{attribute 'qualified_only'}
VAR_GLOBAL
    {attribute 'TcLinkTo' := 'TIID^Device 1 (EtherCAT)^B940_009_R19_DRL_02_E0_EK1200^R19_DRL_02_E4_EK1122^Term 35 (EK1100)^B950-100H1-R02-PNL-01_E2^Channel 1^Input'}
    {attribute 'pytmc' := '
        pv: "DREAM:SL:STATUS",
        field: "DREAM Safety Loop Status",
        field: "ZNAM OPEN",
        field: "ONAM CLOSED"
    '}
    bSafetyLoopStatus AT %I* : BOOL;

        {attribute 'TcLinkTo' := 'TIID^Device 1 (EtherCAT)^B940_009_R19_DRL_02_E0_EK1200^R19_DRL_02_E4_EK1122^Term 35 (EK1100)^B950-100H1-R02-PNL-01_E1^Channel 1^Output'}
    {attribute 'pytmc' := '
        pv: "DREAM:SL:ENABLE",
        field: "DREAM Safety Loop Enable",
        field: "ZNAM OPEN",
        field: "ONAM CLOSED"
    '}
    bSafetyLoopEnable AT %Q*: BOOL;
END_VAR

(* stored: Version 1.1.0.1
   GVL GVL_EPS: Id {b258de69-c58b-428f-a6a3-19396b4a91a6} *)
